FUNCTION_BLOCK FB_OPC_Cell_Unit_4 //EXTENDS FB_OPC_Basic IMPLEMENTS ITF_OPC_Basic
VAR_OUTPUT
	{attribute 'OPC.UA.DA':='1'}
	{attribute 'OPC.UA.DA.Access' := '1'}
	{attribute 'OPC.UA.DA.Description' := 'Cell 4 bridge output data'}
	{attribute 'OPC.UA.DA.DisplayName' := 'Cell 4 bridge output data'}
	{attribute 'OPC.UA.DA.StructuredType' := '1'}
	Output			: ST_Output;

END_VAR
VAR_OUTPUT PERSISTENT
	{attribute 'OPC.UA.DA':='1'}
	{attribute 'OPC.UA.DA.Access' := '3'}
	{attribute 'OPC.UA.DA.Description' := 'Cell 4 bridge input data'}
	{attribute 'OPC.UA.DA.DisplayName' := 'Cell 4 bridge input data'}
	{attribute 'OPC.UA.DA.StructuredType' := '1'}
	Input			: ST_Input;

END_VAR
VAR
	bInitDone					: BOOL;
	bInhibitOPCUpdate			: BOOL;		// Set to TRUE to stop updating values from OPC structures
END_VAR

// Init values
M_Init();

// Data change status handling for cell
IF (NOT Input.Cell.AdditionalData.Settings.DataChangeStatusModeStateEnable) THEN
	Input.Cell.AdditionalData.MESHandShakes.DataChangeStatusModeState := Output.Cell.ModeState.DataChange;
END_IF
IF (NOT Input.Cell.AdditionalData.Settings.DataChangeStatusOEEEnable) THEN
	Input.Cell.AdditionalData.MESHandShakes.DataChangeStatusOEE := Output.Cell.OEE.DataChange;
END_IF
IF (NOT Input.Cell.AdditionalData.Settings.DataChangeStatusErrorWarningEnable) THEN
	Input.Cell.AdditionalData.MESHandShakes.DataChangeStatusErrorWarning := Output.Cell.ErrorWarning.DataChange;
END_IF
IF (NOT Input.Cell.AdditionalData.Settings.DataChangeStatusOperationalDataEnable) THEN
	Input.Cell.AdditionalData.MESHandShakes.DataChangeStatusOperationalData := Output.Cell.OperationalData.DataChange;
END_IF
	
// Data change status handling for Station 1
IF (NOT Input.Station.Station1.AdditionalData.Settings.DataChangeStatusModeStateEnable) THEN
	Input.Station.Station1.AdditionalData.MESHandShakes.DataChangeStatusModeState := Output.Station.Station1.ModeState.DataChange;
END_IF
IF (NOT Input.Station.Station1.AdditionalData.Settings.DataChangeStatusJobDataEnable) THEN
	Input.Station.Station1.AdditionalData.MESHandShakes.DataChangeStatusJobData := Output.Station.Station1.JobData.DataChange;
END_IF
IF (NOT Input.Station.Station1.AdditionalData.Settings.DataChangeStatusOEEEnable) THEN
	Input.Station.Station1.AdditionalData.MESHandShakes.DataChangeStatusOEE := Output.Station.Station1.OEE.DataChange;
END_IF
IF (NOT Input.Station.Station1.AdditionalData.Settings.DataChangeStatusErrorWarningEnable) THEN
	Input.Station.Station1.AdditionalData.MESHandShakes.DataChangeStatusErrorWarning := Output.Station.Station1.ErrorWarning.DataChange;
END_IF
IF (NOT Input.Station.Station1.AdditionalData.Settings.DataChangeStatusCurrentConfigurationEnable) THEN
	Input.Station.Station1.AdditionalData.MESHandShakes.DataChangeStatusCurrentConfiguration := Output.Station.Station1.CurrentConfiguration.DataChange;
END_IF
IF (NOT Input.Station.Station1.AdditionalData.Settings.DataChangeStatusUpcomingConfigurationEnable) THEN
	Input.Station.Station1.AdditionalData.MESHandShakes.DataChangeStatusUpcomingConfiguration := Output.Station.Station1.UpcomingConfiguration.DataChange;
END_IF
IF (NOT Input.Station.Station1.AdditionalData.Settings.DataChangeStatusOperationalDataEnable) THEN
	Input.Station.Station1.AdditionalData.MESHandShakes.DataChangeStatusOperationalData := Output.Station.Station1.OperationalData.DataChange;
END_IF

// Data change status handling for Station 1
IF (NOT Input.Transport.AdditionalData.Settings.DataChangeStatusTransportStatusEnable) THEN
	Input.Transport.AdditionalData.MESHandShakes.DataChangeStatusTransportStatus := Output.Transport.Status.DataChange;
END_IF
IF (NOT Input.Transport.AdditionalData.Settings.DataChangeStatusTransportMappingEnable) THEN
	Input.Transport.AdditionalData.MESHandShakes.DataChangeStatusTransportMapping := Output.Transport.Mapping.DataChange;
END_IF

METHOD M_init : BOOL
VAR_INPUT
END_VAR
IF (NOT bInitDone) THEN
	bInitDone := TRUE;
END_IF
END_METHOD

PROPERTY PUBLIC P_bCellLight : BOOL
GET
P_bCellLight := Input.Cell.Control.EnableCellLight;
END_GET
SET
Output.Cell.OperationalData.General.bCellLight := P_bCellLight;
END_SET
END_PROPERTY

PROPERTY PUBLIC P_bDoors : BOOL
SET
Output.Cell.OperationalData.General.bDoors := P_bDoors;
END_SET
END_PROPERTY

PROPERTY PUBLIC P_bEStop : BOOL
GET
P_bEStop := Output.Cell.OperationalData.General.bEStop;
END_GET
SET
Output.Cell.OperationalData.General.bEStop := P_bEStop;
END_SET
END_PROPERTY

PROPERTY P_bLockDoors : BOOL
GET
P_bLockDoors := Input.Cell.Control.LockDoors;
END_GET
END_PROPERTY

PROPERTY P_bResetEStop : BOOL
GET
P_bResetEStop := Input.Cell.Control.ResetEStop;
END_GET
END_PROPERTY

PROPERTY PUBLIC P_bStationCommOK : BOOL
GET
P_bStationCommOK := Output.Cell.OperationalData.General.bStationCommOK;
END_GET
SET
Output.Cell.OperationalData.General.bStationCommOK := P_bStationCommOK;
END_SET
END_PROPERTY

PROPERTY P_bUnlockDoors : BOOL
GET
P_bUnlockDoors := Input.Cell.Control.UnlockDoors;
END_GET
END_PROPERTY

PROPERTY PUBLIC P_iHeartBeat : UINT
GET
P_iHeartBeat := Input.Header.HeartBeat;
END_GET
SET
Output.Header.HeartBeat := P_iHeartBeat;
END_SET
END_PROPERTY

PROPERTY PUBLIC P_rCPUFrequency : REAL
GET
P_rCPUFrequency := Output.Cell.OperationalData.General.rCPUFrequency;
END_GET
SET
Output.Cell.OperationalData.General.rCPUFrequency := P_rCPUFrequency;
END_SET
END_PROPERTY

PROPERTY PUBLIC P_rOSCPULoad : REAL
GET
P_rOSCPULoad := Output.Cell.OperationalData.General.rOSCPULoad;
END_GET
SET
Output.Cell.OperationalData.General.rOSCPULoad := P_rOSCPULoad;
END_SET
END_PROPERTY

PROPERTY PUBLIC P_rPLCCPULoad : REAL
GET
P_rPLCCPULoad := Output.Cell.OperationalData.General.rPLCCPULoad;
END_GET
SET
Output.Cell.OperationalData.General.rPLCCPULoad := P_rPLCCPULoad;
END_SET
END_PROPERTY

PROPERTY PUBLIC P_rPLCCPUTemp : REAL
GET
P_rPLCCPUTemp := Output.Cell.OperationalData.General.rPLCCPUTemp;
END_GET
SET
Output.Cell.OperationalData.General.rPLCCPUTemp := P_rPLCCPUTemp;
END_SET
END_PROPERTY

PROPERTY PUBLIC P_rSafetyCPUTemp : REAL
GET
P_rSafetyCPUTemp := Output.Cell.OperationalData.General.rSafetyCPUTemp;
END_GET
SET
Output.Cell.OperationalData.General.rSafetyCPUTemp := P_rSafetyCPUTemp;
END_SET
END_PROPERTY

PROPERTY PUBLIC P_sPLCMBSerial : STRING
GET

P_sPLCMBSerial := Output.Cell.OperationalData.General.sPLCMBSerial;
END_GET
SET
Output.Cell.OperationalData.General.sPLCMBSerial := P_sPLCMBSerial;
END_SET
END_PROPERTY

PROPERTY PUBLIC P_sPLCSerial : STRING
GET
P_sPLCSerial := Output.Cell.OperationalData.General.sPLCSerial;
END_GET
SET
Output.Cell.OperationalData.General.sPLCSerial := P_sPLCSerial;
END_SET
END_PROPERTY

END_FUNCTION_BLOCK

(* stored: Version 1.1.0.1, ProductVersion 3.1.4024.5
   POU FB_OPC_Cell_Unit_4: Id {4d74fb34-c831-4b88-ab1b-d763a7c598f7}, SpecialFunc None
   Method M_init: Id {6f313a76-2463-4f2b-b7eb-952d3dfcb38d}
   Property P_bCellLight: Id {4fa91b4a-4b9a-45ab-9a63-8fd3dfcd301a}
   Get Get: Id {6584cd07-c318-41f1-9995-465495b08f18}
   Set Set: Id {9434322f-77b6-452e-a831-8b49fad97eb3}
   Property P_bDoors: Id {cb9dafbb-9216-4814-9a28-da9942595914}
   Set Set: Id {5fdea3c3-4d33-48c0-af7d-78f7143898a4}
   Property P_bEStop: Id {350b058e-4e13-4a29-b9e6-0ad151f03770}
   Get Get: Id {7bdbbbdf-be97-4e78-8d7a-1a7bb9a2a39b}
   Set Set: Id {ce21554d-f274-44c7-900e-dfccfd707f12}
   Property P_bLockDoors: Id {3bb44a5e-7ebd-418b-8ab2-3e2d578ec3a7}
   Get Get: Id {ad8c671c-8ab7-4170-b94c-c542a5f785c1}
   Property P_bResetEStop: Id {91068d9d-4e8c-4c67-86d0-39982401fc21}
   Get Get: Id {63e7abcd-3843-4346-a77d-dd78066c01d5}
   Property P_bStationCommOK: Id {091fc529-1f8a-4fa2-bd09-76bad4223958}
   Get Get: Id {40db9b0d-e0d5-4593-9962-fd17bb6960b0}
   Set Set: Id {c3e54d85-b146-499c-aa16-569f2b9f3e8f}
   Property P_bUnlockDoors: Id {b0ecb8c8-8a65-4e16-b19e-047191b041ea}
   Get Get: Id {bcbce038-3d41-4b7a-b572-2289af306807}
   Property P_iHeartBeat: Id {10f72142-3ba4-4e96-a702-aac9a1d28238}
   Get Get: Id {761ad27f-8d40-48c2-9bb0-d5af87022bd8}
   Set Set: Id {e75fdd67-66d5-4b08-b0d9-4744dfc9d9df}
   Property P_rCPUFrequency: Id {17e740b9-626f-477d-890e-56660cb23ba7}
   Get Get: Id {3cf56568-335a-4882-a976-0ea4abf78015}
   Set Set: Id {99ec6272-9aec-4f2b-83db-80aef5848077}
   Property P_rOSCPULoad: Id {f14f4591-08d8-4c73-bb92-dfad259bbece}
   Get Get: Id {81ade830-5f46-47d2-a3a2-98ddb303c4a8}
   Set Set: Id {b764e910-b8ea-4a48-ac7f-81a31250ed1c}
   Property P_rPLCCPULoad: Id {ba56f122-56a6-4d26-8dd7-f97cfccab867}
   Get Get: Id {a41f06db-47c3-46ad-93a0-a42e6725adeb}
   Set Set: Id {6ddedb1e-2df8-4f25-bb28-899f6be911d7}
   Property P_rPLCCPUTemp: Id {c0e114c6-a8cd-481f-9592-c60b837c1671}
   Get Get: Id {423410fb-316c-4d3c-b9c9-b9e0ba8969f2}
   Set Set: Id {8b625dce-8509-476a-a1c8-22b1cba500e9}
   Property P_rSafetyCPUTemp: Id {78cd3f2e-eb07-4798-a54b-a21babfcc389}
   Get Get: Id {6a171e82-4db3-48e9-a2ca-5ac44be5d338}
   Set Set: Id {67f26075-5874-42bc-a5c7-7c3132553685}
   Property P_sPLCMBSerial: Id {03a400ab-616a-44eb-8e3a-d18f1f32db8a}
   Get Get: Id {ea685a61-5322-4e26-b6dd-1c9e18451859}
   Set Set: Id {087dd1c5-e8fb-49e5-aba8-a23b3d08c3b0}
   Property P_sPLCSerial: Id {040ab2e5-db73-4255-8a83-6b4052337d62}
   Get Get: Id {9aa67b5c-4ffb-4504-baf8-ad8b7c009692}
   Set Set: Id {2183e5e5-e35e-432a-b5e9-7e3002b5cf47} *)
